// This function has been automatically generated from the project information.
{attribute 'signature_flag' := '1073741824'}
{attribute 'TcGenerated'}
{attribute 'no-analysis'}
FUNCTION F_GetTitle : WSTRING
VAR_INPUT
	
END_VAR

F_GetTitle := "AUT_Utilities";

END_FUNCTION

(* stored: Version 1.1.0.1
   POU F_GetTitle: Id {cd090806-ff4e-4d7d-8e8e-f82fe247f96b}, SpecialFunc None *)
